Yaskawa INFORM job: yellow_cover_19_07_23_planes_program.JBI

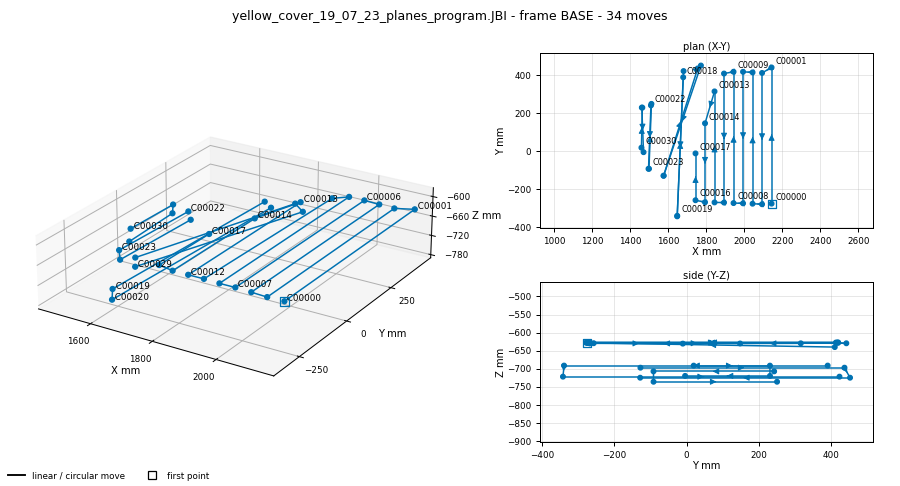
[picture p0: tool path of yellow_cover_19_07_23_planes_program.JBI in frame BASE, 34 of 40 moves have a stored position in this frame; points joined in program order, loops and branches not executed]
/JOB
//NAME yellow_cover_19_07_23_planes_program
//POS
///NPOS 34,0,34,0,0,0
///TOOL 0
///POSTYPE BASE
///RECTAN
///RCONF 0,0,0,0,0,0,0,0,0,0,0,0,0,0,0,0,0,0,0,0,0,0,0,0
C00000=2142.874513,-274.755902,-628.283050,175.000000,-5.000000,5.000000
C00001=2142.874513,441.314098,-629.348050,175.000000,-5.000000,5.000000
C00002=2092.874513,412.481098,-627.386050,175.000000,-5.000000,5.000000
C00003=2092.874513,-277.877902,-627.655050,175.000000,-5.000000,5.000000
C00004=2042.874513,-275.116902,-627.294050,175.000000,-5.000000,5.000000
C00005=2042.874513,415.422098,-627.433050,175.000000,-5.000000,5.000000
C00006=1992.874513,418.527098,-627.273050,175.000000,-5.000000,5.000000
C00007=1992.874513,-273.145902,-626.895050,175.000000,-5.000000,5.000000
C00008=1942.874513,-271.834902,-627.979050,175.000000,-5.000000,5.000000
C00009=1942.874513,418.747098,-627.591050,175.000000,-5.000000,5.000000
C00010=1892.874513,409.378098,-639.818050,175.000000,-5.000000,5.000000
C00011=1892.874513,-269.169902,-628.223050,175.000000,-5.000000,5.000000
C00012=1842.874513,-268.344902,-628.987050,175.000000,-5.000000,5.000000
C00013=1842.874513,315.419098,-629.428050,175.000000,-5.000000,5.000000
C00014=1792.874513,147.737098,-629.908050,175.000000,-5.000000,5.000000
C00015=1792.874513,-267.360902,-629.616050,175.000000,-5.000000,5.000000
C00016=1742.869513,-256.897902,-629.160050,175.000000,-5.000000,5.000000
C00017=1742.869513,-10.568602,-630.317050,175.000000,-5.000000,5.000000
C00018=1678.158500,389.742510,-690.973675,180.000000,-60.000000,0.000000
C00019=1646.848500,-338.674490,-690.973675,180.000000,-60.000000,0.000000
C00020=1646.398500,-341.662490,-721.565175,180.000000,-60.000000,0.000000
C00021=1680.138500,422.359510,-721.565175,180.000000,-60.000000,0.000000
C00022=1508.548100,241.812870,-706.912550,180.000000,-60.000000,0.000000
C00023=1495.702100,-91.547130,-706.912550,180.000000,-60.000000,0.000000
C00024=1498.155100,-91.387130,-735.628050,180.000000,-60.000000,0.000000
C00025=1511.059100,249.862870,-735.628050,180.000000,-60.000000,0.000000
C00026=1575.391750,-127.651600,-696.772663,180.000000,-60.000000,0.000000
C00027=1754.331750,436.117400,-696.772663,180.000000,-60.000000,0.000000
C00028=1771.301750,451.532400,-724.467663,180.000000,-60.000000,0.000000
C00029=1574.831750,-128.313600,-724.467663,180.000000,-60.000000,0.000000
C00030=1458.453050,19.482825,-691.111355,180.000000,-60.000000,0.000000
C00031=1463.248050,230.242825,-691.111355,180.000000,-60.000000,0.000000
C00032=1460.449050,230.352825,-719.455355,180.000000,-60.000000,0.000000
C00033=1469.614050,-4.187175,-719.455355,180.000000,-60.000000,0.000000
///POSTYPE PULSE
///PULSE
EC00000=0
EC00001=0
EC00002=0
EC00003=0
EC00004=0
EC00005=0
EC00006=0
EC00007=0
EC00008=0
EC00009=0
EC00010=0
EC00011=0
EC00012=0
EC00013=0
EC00014=0
EC00015=0
EC00016=0
EC00017=0
EC00018=0
EC00019=0
EC00020=0
EC00021=0
EC00022=92160
EC00023=92160
EC00024=92160
EC00025=92160
EC00026=184320
EC00027=184320
EC00028=184320
EC00029=184320
EC00030=276480
EC00031=276480
EC00032=276480
EC00033=276480
//INST
///DATE 2023/08/07 14:38
///ATTR SC,RW,RJ
////FRAME BASE
///GROUP1 RB1,ST1
NOP
MOVJ P009 EX000 VJ=15.00
MOVJ C00000 EC00000 VJ=15.0
CALL JOB:SPYON
MOVL C00001 EC00001 V=150.0
MOVL C00002 EC00002 V=150.0
MOVL C00003 EC00003 V=150.0
MOVL C00004 EC00004 V=150.0
MOVL C00005 EC00005 V=150.0
MOVL C00006 EC00006 V=150.0
MOVL C00007 EC00007 V=150.0
MOVL C00008 EC00008 V=150.0
MOVL C00009 EC00009 V=150.0
MOVL C00010 EC00010 V=150.0
MOVL C00011 EC00011 V=150.0
MOVL C00012 EC00012 V=150.0
MOVL C00013 EC00013 V=150.0
MOVL C00014 EC00014 V=150.0
MOVL C00015 EC00015 V=150.0
MOVL C00016 EC00016 V=150.0
MOVL C00017 EC00017 V=150.0
CALL JOB:SPYOF
MOVJ P009 VJ=15.00
MOVJ C00018 EC00018 VJ=15.0
CALL JOB:SPYON
MOVL C00019 EC00019 V=150.0
MOVL C00020 EC00020 V=150.0
MOVL C00021 EC00021 V=150.0
CALL JOB:SPYOF
MOVJ P009 VJ=15.00
MOVJ C00022 EC00022 VJ=15.0
CALL JOB:SPYON
MOVL C00023 EC00023 V=150.0
MOVL C00024 EC00024 V=150.0
MOVL C00025 EC00025 V=150.0
CALL JOB:SPYOF
MOVJ P009 VJ=15.00
MOVJ C00026 EC00026 VJ=15.0
CALL JOB:SPYON
MOVL C00027 EC00027 V=150.0
MOVL C00028 EC00028 V=150.0
MOVL C00029 EC00029 V=150.0
CALL JOB:SPYOF
MOVJ P009 VJ=15.00
MOVJ C00030 EC00030 VJ=15.0
CALL JOB:SPYON
MOVL C00031 EC00031 V=150.0
MOVL C00032 EC00032 V=150.0
MOVL C00033 EC00033 V=150.0
CALL JOB:SPYOF
MOVJ P009 VJ=15.00
END
